// TwinCAT 3 PLC project PLC
// ProgramVersion: 3.1.4024.0
// libraries:
//   Tc2_Standard, * (Beckhoff Automation GmbH)
//   Tc2_System, * (Beckhoff Automation GmbH)
//   Tc3_Module, * (Beckhoff Automation GmbH)
//   VisuDialogs, * (System)
//   VisuSymbols,3.5.10.0,System
// project tree:
//   / GlobalTextList.TcGTLO, PlcTask.TcTTO (not stored), Visualization Manager.TcVMO (not stored)
//   POUs/ FB_Pulse.TcPOU, MAIN.TcPOU, p10_ladder.TcPOU (not stored), p20_timer.TcPOU
//   VISUs/ Visualization.TcVIS

// ---- POUs/FB_Pulse.TcPOU
FUNCTION_BLOCK FB_Pulse
VAR_INPUT
END_VAR
VAR_OUTPUT
END_VAR
VAR
END_VAR

END_FUNCTION_BLOCK

// ---- POUs/MAIN.TcPOU
PROGRAM MAIN
VAR
	bStartMotor : BOOL := FALSE;
	bStopMotor  : BOOL := FALSE;
	bServoMotor : BOOL;
	sr_MotorSetReset : SR;
END_VAR


sr_MotorSetReset(SET1:= bStartMotor,
				 RESET:= bStopMotor,
				 Q1 => bServoMotor);

p10_ladder();

END_PROGRAM

// ---- POUs/p20_timer.TcPOU
PROGRAM p20_timer
VAR
END_VAR

END_PROGRAM

// ---- GlobalTextList.TcGTLO
TEXTLIST GlobalTextList
  288 = 'Start'
  446 = 'Stop'
END_TEXTLIST

// ---- VISUs/Visualization.TcVIS
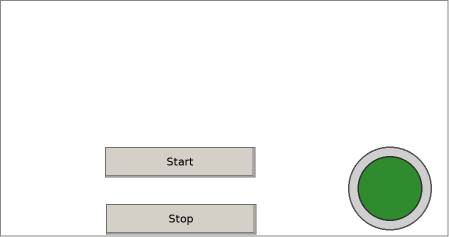
VISUALIZATION Visualization  // 449x237
    Button (105,147 150x30), "Start"
        OnMouseDown: execute { MAIN.bStartMotor := TRUE; }
        OnMouseUp: execute { MAIN.bStartMotor :=  FALSE; }
    Button (106,204 150x30), "Stop", pressed state: MAIN.bStopMotor
        OnMouseDown: execute { MAIN.bStopMotor := TRUE; }
        OnMouseUp: execute { MAIN.bStopMotor := FALSE; }
    Lamp1 (331,140 118x97), variable: MAIN.bServoMotor, style: Lamp-Lamp1-Green
END_VISUALIZATION
